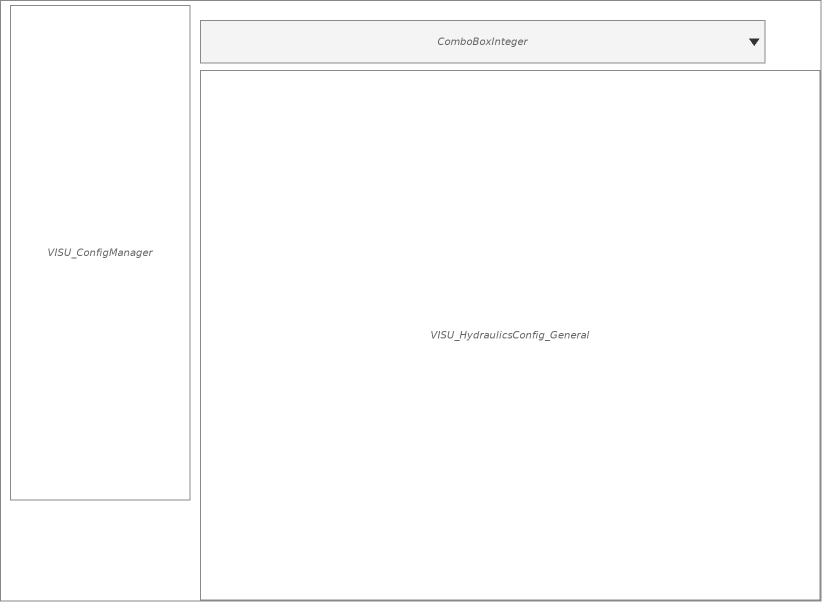
VISUALIZATION VISU_HydraulicsConfig  // 822x602
VAR_IN_OUT
    editable : HydraulicsConfig;
	active : HydraulicsConfig;
    mgr : ConfigManager;
    mgrWidget : ConfigManagerWidget;
    widget : HydraulicsWidget;
END_VAR
    Frame (10,5 180x495)
        shows VISU_ConfigManager(mgr := mgr, widget := mgrWidget)
    ComboBoxInteger (200,20 565x43), variable: widget.activeConfigTab, text list: 'HydraulicsConfigTabsTextList'
    Frame (200,70 620x530), frame switch variable: widget.activeConfigTab
        shows VISU_HydraulicsConfig_General(editable := editable, active := active)
        shows VISU_HydraulicsConfig_Side_General(editable := editable.top, active := active.top)
        shows VISU_MeasurementConfig(active := active.top.pressureMeasurement, editable := editable.top.pressureMeasurement)
        shows VISU_MeasurementConfig(active := active.top.frequencyMeasurement, editable := editable.top.frequencyMeasurement)
        shows VISU_HydraulicsConfig_Side_General(editable := editable.bottom, active := active.bottom)
        shows VISU_MeasurementConfig(active := active.bottom.pressureMeasurement, editable := editable.bottom.pressureMeasurement)
        shows VISU_MeasurementConfig(active := active.bottom.frequencyMeasurement, editable := editable.bottom.frequencyMeasurement)
END_VISUALIZATION

(* stored: Version 1.1.0.1, ProductVersion 3.1.4019.2
   Visu VISU_HydraulicsConfig: Id {a3c39255-3769-48f2-90b9-98901ce80e7a} *)
